# EPICS autosave request: GalilSup/Db/galil_analog_out.req
$(P)$(R)_SP.VAL
$(P)$(R)_SP.DESC
$(P)$(R)_MON.DESC
$(P)$(R)Deadb_SP.VAL
